{attribute 'qualified_only'}
{attribute 'global_init_slot' := '40505'}
VAR_GLOBAL
	fbPodzespoltestowy1						: FB_TestowyPodzespol;
	fbPodzespoltestowy2						: FB_TestowyPodzespol;
	fbPodzespoltestowy3						: FB_TestowyPodzespol;
END_VAR

(* stored: Version 1.1.0.1, ProductVersion 3.1.4024.11
   GVL GVL_Podzespoly: Id {eb9fd0a3-8436-4931-a171-7c6dca862309} *)
